// TRUE for STRING and WSTRING.
//
// Split out so the rule lives in one place: 'is this a string' is asked by the
// comparison, by the formatter, and eventually by the reporters when they decide
// whether a value needs quoting.
FUNCTION TestValueIsText : BOOL
VAR_INPUT
	Value : ANY;
END_VAR

TestValueIsText := (Value.TypeClass = __SYSTEM.TYPE_CLASS.TYPE_STRING)
				OR (Value.TypeClass = __SYSTEM.TYPE_CLASS.TYPE_WSTRING);

END_FUNCTION

(* stored: Version 1.1.0.1, ProductVersion 3.1.4026.0
   POU TestValueIsText: Id {0cb71660-9023-4bfd-8e2b-a8b5641d516d}, SpecialFunc None *)
